FUNCTION_BLOCK FB_Scale
VAR_INPUT	
	diInPutToScale			:DINT; // Värde som ska skalas
	diX0StarterValScaled	:DINT; // Startvärde, tex 0
	diX1EndValScaled		:DINT; // Slutvärde, tex 1000
	diY0StartOut			:DINT; // Startvärde skalat
	iY1EndOut				:DINT; // Slutvärde skalat
END_VAR
VAR_OUTPUT
	diOutPutVal				:DINT; // Utvärde
END_VAR

IF diX1EndValScaled > 0 AND diX1EndValScaled > diX0StarterValScaled  THEN 
	diOutPutVal := (diInPutToScale - diX0StarterValScaled) * (iY1EndOut - diY0StartOut) / (diX1EndValScaled - diX0StarterValScaled) + iY1EndOut;
	ELSE diOutPutVal := 0;
END_IF

END_FUNCTION_BLOCK

(* stored: Version 1.1.0.1, ProductVersion 3.1.4024.11
   POU FB_Scale: Id {95e40287-3797-4ad8-81a3-e0341602b233}, SpecialFunc None *)
